FUNCTION_BLOCK Timer
  (* Standard: 61499-2 *)
  (* Version 0.1, 2015-00-04, SYY, SYY-PC *)
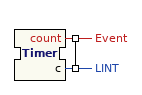
  EVENT_OUTPUT
    count WITH c;
  END_EVENT
  VAR_OUTPUT
    c : LINT := 0;
  END_VAR
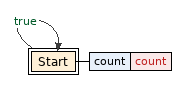
  EC_STATES
    Start : count -> count;
  END_STATES
  EC_TRANSITIONS
    Start TO Start := true;
  END_TRANSITIONS
  ALGORITHM count IN C:
me->c=me->c+1;
  END_ALGORITHM
END_FUNCTION_BLOCK
